# EPICS IOC start-up script: iocsh/gjsAxis.iocsh
# We don't have that comand yet
# The controller currently creates all axes
#gjsCreateAxis("$(MOTOR_PORT)", "$(AXIS_NO)")

dbLoadRecords("./db/gjsmotor.template", "PREFIX=$(PREFIX), MOTOR_NAME=$(MOTOR_NAME), AXIS_NO=$(AXIS_NO), R=$(MOTOR_NAME)-, MOTOR_PORT=$(MOTOR_PORT), ASYN_PORT=$(ASYN_PORT), AXIS_NO=$(AXIS_NO), DESC=$(DESC), PREC=$(PREC), SREV=$(SREV), UREV=$(UREV), DHLM=$(DHLM), DLLM=$(DLLM)")
